(* IEC 61131-3 sources: AXOpen/src/components.rexroth.drives/ctrl/src/AxoCtrlxDriveXsc/TypesStructuresAndEnums, 22 files *)

(* ---- AxoCtrlxDriveXscErrorStruct.st ---- *)
NAMESPACE AXOpen.Components.Rexroth.Drives
    TYPE
        {S7.extern=ReadWrite}
        AxoCtrlxDriveXscErrorStruct :
        STRUCT
            Table       : AXOpen.Components.Rexroth.Drives.eAxoCtrlxDriveXscErrorTable;          (* Additional diagnosis table           *)
            Additional1 : DWORD;                (* Additional diagnosis number1         *)
            Additional2 : DWORD;                (* Additional diagnosis number2         *)
        END_STRUCT;
    END_TYPE
END_NAMESPACE

(* ---- eAxoCtrlxDriveXscErrorCode.st ---- *)
NAMESPACE AXOpen.Components.Rexroth.Drives
    TYPE PUBLIC
        eAxoCtrlxDriveXscErrorCode : WORD
        (
            NONE_ERROR                  := WORD#16#0000,     (* No error code available              *)
            (*                  invalid input                                                   *)
            INPUT_INVALID_ERROR         := WORD#16#0001,     (* Invalid input                        *)
            (*                  communications error                                            *)
            COMMUNICATION_ERROR         := WORD#16#0002,     (* Error while communication            *)
            (*                  data processing error                                           *)
            RESOURCE_ERROR              := WORD#16#0003,     (* Resource error                       *)
            ACCESS_ERROR                := WORD#16#0004,     (* Access error                         *)
            STATE_MACHINE_ERROR         := WORD#16#0005,     (* Invalid state State - Machine        *)
            INPUT_RANGE_ERROR           := WORD#16#0006,     (* Error because Input out of range     *)
            CALCULATION_ERROR           := WORD#16#0007,     (* Error while calculation              *)
            (*                  device error                                                    *)
            DEVICE_ERROR                := WORD#16#0008,     (* Device Error occurred                *)
            (*                  other error                                                     *)
            OTHER_ERROR                 := WORD#16#7FFE,     (* Undefined Error                      *)
            (*                  system error                                                    *)
            SYSTEM_ERROR                := WORD#16#7FFF      (* System error occured                 *)

                );
    END_TYPE
END_NAMESPACE

(* ---- eAxoCtrlxDriveXscErrorTable.st ---- *)
NAMESPACE AXOpen.Components.Rexroth.Drives
    TYPE PUBLIC
        eAxoCtrlxDriveXscErrorTable : WORD
        (
            NO_TABLE_USED           := WORD#16#0000,         //reserved
            SERCOS_TABLE            := WORD#16#0010,         //Sercos Error: Addtitional1 = Sercos Code
            MLDS_TABLE              := WORD#16#0020,         //Drive-based Motion - Logic
            MLC_TABLE               := WORD#16#0030,         //Controller - based Motion - Logic
            MTX_TABLE               := WORD#16#0040,         //CNC
            MLP_TABLE               := WORD#16#0050,         //PC  - based Motion Logic
            PLC_TABLE               := WORD#16#0060,         //PLC
            INDRV_TABLE             := WORD#16#0070,         //IndraDrive
            DIAX_TABLE              := WORD#16#0080,         //DIAX
            ECO_TABLE               := WORD#16#0090,         //EcoDrive
            PB_DP_TABLE             := WORD#16#0130,         //Profibus
            DEVICENET_TABLE         := WORD#16#0140,         //DeviceNet
            ETHERNET_TABLE          := WORD#16#0150,         //Ethernet
            INTERBUS_TABLE          := WORD#16#0160,         //Interbus
            F_RELATED_TABLE         := WORD#16#0170,         //function related
            USER1_TABLE             := WORD#16#1000,         //free User Table
            USER2_TABLE             := WORD#16#1001,         //free User Table
            USER3_TABLE             := WORD#16#1002,         //free User Table
            USER4_TABLE             := WORD#16#1003,         //free User Table
            USER5_TABLE             := WORD#16#1004,         //free User Table
            USER6_TABLE             := WORD#16#1005,         //free User Table
            USER7_TABLE             := WORD#16#1006,         //free User Table
            USER8_TABLE             := WORD#16#1007,         //free User Table
            USER9_TABLE             := WORD#16#1008,         //free User Table
            USER10_TABLE            := WORD#16#1009          //free User Table
        );
    END_TYPE
END_NAMESPACE

(* ---- AxoCtrlxDriveXsc_Component_Status.st ---- *)
NAMESPACE AXOpen.Components.Rexroth.Drives
    {S7.extern=ReadWrite}
    {#ix-attr:[Container(Layout.Stack)]}
    CLASS PUBLIC AxoCtrlxDriveXsc_Component_Status EXTENDS AXOpen.Components.Abstractions.AxoComponent_Status
        VAR PUBLIC

        END_VAR
    END_CLASS
END_NAMESPACE

(* ---- AxoCtrlxDriveXsc_Config.st ---- *)
NAMESPACE AXOpen.Components.Rexroth.Drives
    {S7.extern=ReadWrite}
    {#ix-attr:[Container(Layout.Stack)]}
    CLASS PUBLIC AxoCtrlxDriveXsc_Config
        VAR PUBLIC
            {#ix-set:AttributeName = "<#Info time#>"}
            InfoTime : LTIME := LT#5S;
            {#ix-set:AttributeName = "<#Error time#>"}
            ErrorTime : LTIME := LT#10S;
        END_VAR
    END_CLASS
END_NAMESPACE

(* ---- AxoCtrlxDriveXsc_Control.st ---- *)
NAMESPACE AXOpen.Components.Rexroth.Drives
    {S7.extern=ReadWrite}
    {#ix-attr:[Container(Layout.Stack)]}
    CLASS PUBLIC AxoCtrlxDriveXsc_Control
        VAR PUBLIC

        END_VAR
    END_CLASS
END_NAMESPACE

(* ---- AxoCtrlxDriveXsc_In.st ---- *)
NAMESPACE AXOpen.Components.Rexroth.Drives
    {S7.extern=ReadWrite}
    {#ix-attr:[Container(Layout.Wrap)]}
    CLASS PUBLIC AxoCtrlxDriveXsc_In
        VAR PUBLIC
            {#ix-set:AttributeName = "<#Status#>"}
            {#ix-attr:[ReadOnly()]}
            Status           :   AxoCtrlxDriveXsc_Status;
        END_VAR
    END_CLASS
END_NAMESPACE

(* ---- AxoCtrlxDriveXsc_Out.st ---- *)
NAMESPACE AXOpen.Components.Rexroth.Drives
    {S7.extern=ReadWrite}
    {#ix-attr:[Container(Layout.Wrap)]}
    CLASS PUBLIC AxoCtrlxDriveXsc_Out
        VAR PUBLIC
            {#ix-set:AttributeName = "<#Control#>"}
            {#ix-attr:[ReadOnly()]}
            Control           :   AxoCtrlxDriveXsc_Control;
        END_VAR
    END_CLASS
END_NAMESPACE

(* ---- AxoCtrlxDriveXsc_Status.st ---- *)
NAMESPACE AXOpen.Components.Rexroth.Drives
    {S7.extern=ReadWrite}
    {#ix-attr:[Container(Layout.Stack)]}
    CLASS PUBLIC AxoCtrlxDriveXsc_Status
        VAR PUBLIC

        END_VAR
    END_CLASS
END_NAMESPACE

(* ---- AxoCtrlxDriveXscAxisData.st ---- *)
NAMESPACE AXOpen.Components.Rexroth.Drives
    {S7.extern=ReadWrite}
    CLASS AxoCtrlxDriveXscAxisData
        VAR PUBLIC
            (* Commands *)
            CallAxis					:	BOOL;			//Call axis method for cyclic communication
            ReadOnlyData				:	BOOL;			//Read only data values from drive
            CallNumberCyclic			:	INT :=-1; 		//Number of method call's for cyclic communication
            WriteCommand				:	BOOL;			//Write command to drive
            PowerOnReq					:	BOOL;			//Request to power the drive on
            ResetReq					:	BOOL;			//Request to reset the drive
            HomingReq					:	BOOL;			//Request to start homing
            JogPositiveReq				:	BOOL;			//Request to jog the drive in positive direction
            JogNegativeReq				:	BOOL;			//Request to jog the drive in negative direction
            DriveStopReq				:	BOOL;			//Set Drive Stop with writing deceleration value to drive
            DriveHaltReq				:	BOOL;			//Set Drive Halt with writing deceleration value to drive
            MoveVelocityReq				:	BOOL;			//Command is velocity
            TorqueControlReq				:	BOOL;			//Command is torque
            Relative					:	BOOL; 			//Move relative to (last recommended) positioning command value
            Additive					:	BOOL; 			//Move additive to actual position; works only if relative possitioning active
            Position					:	LREAL;			//Target position for the motion  (negative or positive)
            Velocity					:	LREAL;			//Value of the maximum velocity (always positive) (not necessarily reached) [u/s].
            Acceleration				:	LREAL;			//Value of the acceleration (always positive) (increasing energy of the motor) [u/s2]
            Deceleration				:	LREAL;			//Value of the deceleration (always positive) (decreasing energy of the motor) [u/s2]
            Jerk						:	LREAL;			//Value of the jerk (always positive) [u/s3]
            Torque						:	LREAL;			//Value of the torque (always positive)
            S_0_0144_SignalStateWord	: 	WORD;			//S-0-0144 SignalStateWord*)
            CallAxisParameterMethod		:	BOOL;			//Call axis method for parameter read/write
            EnableAcyclicCommunication	:	BOOL;			//Enable acyclic communication (for parameter read/write)
            CallNumberAcyclic			:	INT;			//Number of method call's for acyclic communication
            WriteParameter				:	BOOL;			//FALSE = read, TRUE  = write Value of selected Parameter
            SelectDataType				:	UINT;			//0= Bool, 1 = Any, 2 = REAL
            ParameterNumber				:	DINT;			//Parameter number
            WriteValueLint				:	LINT;			//DINT value to be written
            WriteValueReal				:	REAL;			//REAL value to be written
            OverrideVelocityFactor		:	LREAL := 1.0;	//LREAL value to be written
            OverrideAccelerationFactor	:	LREAL := 1.0;	//LREAL value to be written
            OverrideJerkFactor			:	LREAL := 1.0;	//LREAL value to be written
        (* States *)
            CommandWriteActive			:	BOOL; 			//Command transfer to drive is active
            SetpointReached				: 	BOOL;			//Setpoint reached
            PowerOK						:	BOOL; 			//Power OK
            HomeOK						:	BOOL;			//Drive has reached the homeposition
            ResetOK						:	BOOL; 			//Reset done
            HomingRunning				:	BOOL;			//Homing is active
            Stopped						:	BOOL; 			//Drive in stopped regularly
            Standstill					:	BOOL; 			//Drive in standstill
            InPosition					:	BOOL; 			//Drive in position
            StoppedDueError				:	BOOL; 			//Drive in stop due to error
            MessageActive				:	BOOL;			//Class 3 diagnostics (message) present
            WarningActive				:	BOOL;			//Class 2 diagnostics (warning) present
            FailureActive				:	BOOL;			//Class 1 diagnostics (failure) present
            PowerError					:	BOOL; 			//Power-Failure
            StopError					:	BOOL;			//Stopping-Failure
            ContinuousMotion			:	BOOL; 			//Continius motion
            DiscreteMotion				:	BOOL; 			//Discrete motion
            SynchronizedMotion			:	BOOL;			//Synchronized motion
            Error						:	BOOL;			//Error
            ErrorID						:	AXOpen.Components.Rexroth.Drives.eAxoCtrlxDriveXscErrorCode;		//Error identification, ErrorCode
            ErrorIdent					:	AXOpen.Components.Rexroth.Drives.AxoCtrlxDriveXscErrorStruct;	//Error identification
            ActualPosition				:	LREAL; 			//Shows actual position
            ActualVelocity				:	LREAL; 			//Shows actual velocity
            ActualTorque				:	LREAL; 			//Shows actual torque
            CheckAccessOK				:	BOOL := TRUE;	//Flag for checking valid access at Axis_Data array
            S_0_0145_SignalControlWord	:	WORD;			//S-0-0145 wSignalControlWord, **** exept bit 0 *****)

            DoneAcyclicCommunication 	:	BOOL; 			//Reading/writing of the individual parameter completed, output variables valid
            ActiveAcyclicCommunication	: 	BOOL; 			//Reading/writing of the individual parameter active, output variables invalid
            DecimalPlaces 				:	UINT;			//Decimal places of the selected parameters
            DataTypeRead				:	UINT; 			//Read data type of the selected parameters
            DataLengthRead				:	UINT;			//Length of the read parameters
            ReadValueDint				:	DINT;			//DINT Operating value of the individual parameter without weighting
            ReadValueReal				:	REAL;			//REAL weighted operating value
            Error_AcyclicCommunication	:	BOOL := FALSE;  //Error
            ErrorID_AcyclicCommunication:   AXOpen.Components.Rexroth.Drives.eAxoCtrlxDriveXscErrorCode;		//Error identification, ErrorCode
            ErrorIdent_AcyclicCommunication:AXOpen.Components.Rexroth.Drives.AxoCtrlxDriveXscErrorStruct; 	//Error identification
            hwID                :   WORD;
            hwIdParamCh_IDN     :   WORD;
            hwIdInput_9_Words   :   WORD;
            hwIdOutput_13_Words :   WORD;
        END_VAR
    END_CLASS
END_NAMESPACE

(* ---- AxoCtrlxDriveXscAxisReference.st ---- *)
// USING AXOpen.Components.Drives;

NAMESPACE AXOpen.Components.Rexroth.Drives
    {S7.extern=ReadWrite}
    CLASS AxoCtrlxDriveXscAxisReference IMPLEMENTS AXOpen.Components.Abstractions.Drives.IAxoAxisReference
        VAR PUBLIC
            FieldBus_In     :   AXOpen.Components.Rexroth.Drives.AxoCtrlxDriveXscFieldBusIn;
            FieldBus_Out    :   AXOpen.Components.Rexroth.Drives.AxoCtrlxDriveXscFieldBusOut;
            Parameter_In    :   AXOpen.Components.Rexroth.Drives.AxoCtrlxDriveXscParameterIn;
            Parameter_Out   :   AXOpen.Components.Rexroth.Drives.AxoCtrlxDriveXscParameterOut;
            Data            :   AXOpen.Components.Rexroth.Drives.AxoCtrlxDriveXscAxisData;
            Config          :   AXOpen.Components.Drives.AxoDrive_Config;
            Status          :   AXOpen.Components.Drives.AxoDrive_Status;
        END_VAR
    END_CLASS
END_NAMESPACE

(* ---- AxoCtrlxDriveXscDriveControlWord_S_0_0134_0_0.st ---- *)
NAMESPACE AXOpen.Components.Rexroth.Drives
    {S7.extern=ReadWrite}
    {#ix-attr:[Container(Layout.Wrap)]}
    {#ix-attr:[Group(GroupLayout.GroupBox)]}
    {#ix-set:AttributeName = "<#DriveControlWord#>"}
    CLASS AxoCtrlxDriveXscDriveControlWord_S_0_0134_0_0
        VAR PUBLIC
            {#ix-set:AttributeName = "<#_bit00_Reserve#>"}
            {#ix-attr:[ReadOnly()]}
            _bit00_Reserve 				:	BOOL;
            {#ix-set:AttributeName = "<#_bit01_Reserve#>"}
            {#ix-attr:[ReadOnly()]}
            _bit01_Reserve 				:	BOOL;
            {#ix-set:AttributeName = "<#_bit02_Reserve#>"}
            {#ix-attr:[ReadOnly()]}
            _bit02_Reserve 				:	BOOL;
            {#ix-set:AttributeName = "<#_bit03_Reserve#>"}
            {#ix-attr:[ReadOnly()]}
            _bit03_Reserve 				:	BOOL;
            {#ix-set:AttributeName = "<#_bit04_Reserve#>"}
            {#ix-attr:[ReadOnly()]}
            _bit04_Reserve 				:	BOOL;
            {#ix-set:AttributeName = "<#_bit05_Reserve#>"}
            {#ix-attr:[ReadOnly()]}
            _bit05_Reserve 				:	BOOL;
            {#ix-set:AttributeName = "<#_bit06_Reserve#>"}
            {#ix-attr:[ReadOnly()]}
            _bit06_Reserve 				:	BOOL;
            {#ix-set:AttributeName = "<#_bit07_Reserve#>"}
            {#ix-attr:[ReadOnly()]}
            _bit07_Reserve 				:	BOOL;

            {#ix-set:AttributeName = "<#Command operation mode Bit 0#>"}
            {#ix-attr:[ReadOnly()]}
            CommandOperationModeBit0 	:	BOOL;		//  Command operation mode bit 0                        |   000:  Primary operation mode
                                                        //                                                      |   001:  Secondary operation mode 1
            {#ix-set:AttributeName = "<#Command operation mode Bit 1#>"}
            {#ix-attr:[ReadOnly()]}
            CommandOperationModeBit1 	:	BOOL;		//  Command operation mode bit 1                        |   010:  Secondary operation mode 2
                                                        //                                                      |   011:  Secondary operation mode 3
                                                        //                                                      |   100:  Secondary operation mode 4
            {#ix-set:AttributeName = "<#Command operation mode Bit 2#>"}
            {#ix-attr:[ReadOnly()]}
            CommandOperationModeBit2 	:	BOOL;		//  Command operation mode bit 2                        |   101:  Secondary operation mode 5
                                                        //                                                      |   110:  Secondary operation mode 6
                                                        //                                                      |   111:  Secondary operation mode 7
            {#ix-set:AttributeName = "<#_bit11_Reserve#>"}
            {#ix-attr:[ReadOnly()]}
            _bit11_Reserve 				:	BOOL;
            {#ix-set:AttributeName = "<#_bit12_Reserve#>"}
            {#ix-attr:[ReadOnly()]}
            _bit12_Reserve 				:	BOOL;
            {#ix-set:AttributeName = "<#Drive Halt#>"}
            {#ix-attr:[ReadOnly()]}
            DriveHalt 				:	BOOL;		        //  1-0 change: Deceleration of drive while maintaining maximum acceleration (S‑0‑0138 - only possible if bits 14 and 15 = 1)
            {#ix-set:AttributeName = "<#Drive enable#>"}
            {#ix-attr:[ReadOnly()]}
            DriveEnable 				:	BOOL;		    //  Negative edge: Torque disable without delay (independent of bit 15 or 13)
            {#ix-set:AttributeName = "<#Drive On#>"}
            {#ix-attr:[ReadOnly()]}
            DriveOn 				:	BOOL;		        //  Negative edge: Best possible deceleration (only possible if bit 14 = 1)
        END_VAR
    END_CLASS
END_NAMESPACE

(* ---- AxoCtrlxDriveXscDriveStatusWord_S_0_0135_0_0.st ---- *)
NAMESPACE AXOpen.Components.Rexroth.Drives
    {S7.extern=ReadWrite}
    {#ix-attr:[Container(Layout.Wrap)]}
    {#ix-attr:[Group(GroupLayout.GroupBox)]}
    {#ix-set:AttributeName = "<#DriveStatusWord#>"}
    CLASS AxoCtrlxDriveXscDriveStatusWord_S_0_0135_0_0
        VAR PUBLIC
            {#ix-set:AttributeName = "<#_bit00_Reserve#>"}
            // {#ix-attr:[ReadOnly()]}
            _bit00_Reserve 				:	BOOL;
            {#ix-set:AttributeName = "<#_bit01_Reserve#>"}
            // {#ix-attr:[ReadOnly()]}
            _bit01_Reserve 				:	BOOL;
            {#ix-set:AttributeName = "<#_bit02_Reserve#>"}
            // {#ix-attr:[ReadOnly()]}
            _bit02_Reserve 				:	BOOL;
            {#ix-set:AttributeName = "<#CommandProcessingStatus#>"}
            // {#ix-attr:[ReadOnly()]}
            CommandProcessingStatus		:	BOOL;		//  0 - Drive ignores command value input           |   1 -Drive follows command value input
            {#ix-set:AttributeName = "<#InStandstill#>"}
            // {#ix-attr:[ReadOnly()]}
            InStandstill 				:	BOOL;		//  Drive "Halt" status                             |   1- Act vel < standstill window
            {#ix-set:AttributeName = "<#InReference#>"}
            // {#ix-attr:[ReadOnly()]}
            InReference 				:	BOOL;		//  Drive hommed
            {#ix-set:AttributeName = "<#_bit06_Reserve#>"}
            // {#ix-attr:[ReadOnly()]}
            _bit06_Reserve 				:	BOOL;
            {#ix-set:AttributeName = "<#HardwareLock#>"}
            // {#ix-attr:[ReadOnly()]}
            HardwareLock                :	BOOL;       //  Hardware lock (E-stop)
            {#ix-set:AttributeName = "<#ActualOperatingModeBit0#>"}
            // {#ix-attr:[ReadOnly()]}
            ActualOperatingModeBit0 	:	BOOL;		//  Actual_operating mode bit 0                     |   000:  Primary operation mode
                                                        //                                                  |   001:  Secondary operation mode 1
            {#ix-set:AttributeName = "<#ActualOperatingModeBit1#>"}
            // {#ix-attr:[ReadOnly()]}
            ActualOperatingModeBit1 	:	BOOL;		//  Actual_operating mode bit 1                     |   010:  Secondary operation mode 2
                                                        //                                                  |   011:  Secondary operation mode 3
                                                        //                                                  |   100:  Secondary operation mode 4
            {#ix-set:AttributeName = "<#ActualOperatingModeBit2#>"}
            // {#ix-attr:[ReadOnly()]}
            ActualOperatingModeBit2 	:	BOOL;		//  Actual_operating mode bit 2                     |   101:  Secondary operation mode 5
                                                        //                                                  |   110:  Secondary operation mode 6
                                                        //                                                  |   111:  Secondary operation mode 7
            {#ix-set:AttributeName = "<#_bit11_Reserve#>"}
            // {#ix-attr:[ReadOnly()]}
            _bit11_Reserve 				:	BOOL;
            {#ix-set:AttributeName = "<#WarningZKL2#>"}
            // {#ix-attr:[ReadOnly()]}
            WarningZKL2 				:	BOOL;		//  Warning ZKL2
            {#ix-set:AttributeName = "<#DriveErrorZKL1#>"}
            // {#ix-attr:[ReadOnly()]}
            DriveErrorZKL1 				:	BOOL;		//  Drive Error ZKL1
            {#ix-set:AttributeName = "<#ReadyForOperation Bit 0#>"}
            // {#ix-attr:[ReadOnly()]}
            ReadyForOperationBit0       :	BOOL;		//  Ready to operate bit 0 lower significant bit    |   10: Control section and power section ready for op. (Ab)
                                                        //                                                  |   11: In operation, with torque (e.g. AF)
            {#ix-set:AttributeName = "<#ReadyForOperation Bit 1#>"}
            // {#ix-attr:[ReadOnly()]}
            ReadyForOperationBit1       :	BOOL;		//  Ready to operate bit 1 higher significant bit   |   00: Not ready for power on (e.g., P2)
                                                        //                                                  |   01: Ready for power on (bb)
        END_VAR
    END_CLASS
END_NAMESPACE

(* ---- AxoCtrlxDriveXscFieldBusIn.st ---- *)
NAMESPACE AXOpen.Components.Rexroth.Drives
    {S7.extern=ReadWrite}
    CLASS AxoCtrlxDriveXscFieldBusIn
        (******************* Drive configuration  ***********************
        Master communication; Fieldbus settings:
                Parameter channel 10Bytes / 5 Words I/O
                Parameter channel: F-Modul not used
                Realtime Input channel 18Bytes / 9 Words I/O
                Realtime Output channel 26Bytes / 13 Words I/O
                Profile type: * free configurable mode*
                    Configuration of realtime channel:
                        realtime input (configured feedback values):	    (9words)
                                P-0-4078 Fieldbus status WORD               (2bytes)
                                S-0-0051 Position feedback 1 value          (4bytes)
                                S-0-0040 Veloccity feedback value           (4bytes)
                                S-0-0390 Diagnostig message number          (4bytes)
                                S-0-0144 Signal status  word			    (2bytes)
                                S-0-0084 Actual torque/force value          (2bytes)
                        realtime output (configured command values):		(13words)
                                P-0-4077 Fieldbus control WORD              (2bytes)
                                S-0-0282 Positioning command value          (4bytes)
                                S-0-0259 Positioning velocity value         (4bytes)
                                S-0-0260 Positioning Accelelration          (4bytes)
                                S-0-0359 Positioning Deceleration           (4bytes)
                                S-0-0145 Signal control word                (2bytes)
                                S-0-0080 Torque/force command value		    (2bytes)
                                S-0-0193 Positioning jerk                   (4bytes)
                General settings:
                        S-0-0027, Configuration list signal control word -> Number 0; Content S-0-0393
                        S-0-0329, Assign list signal control word -> Number 0; Content 2
                        Primary operation mode: Drive controlled positioning, encoder 1 (without axis control word)
                        Secondary operation mode: Torque/force control
        *)
        VAR PUBLIC
            PhaseAcknowledgeBit0		:	BOOL;		//Operating mode acknowledge bit 0
            PhaseAcknowledgeBit1 		:	BOOL;		//Operating mode acknowledge bit 1
            InReference 				:	BOOL;		//In reference
            InStandstill 				:	BOOL;		//In standstill
            SetpointReached				:	BOOL;		//Setpoint reached
            CommandChangeBit 			:	BOOL;		//Command change bit
            OperatingModeError 			:	BOOL;		//Operating mode_error
            StatusSetpointProcess 		:	BOOL;		//Status setpoint processing
            ActualOperatingModeBit0 	:	BOOL;		//Actual_operating mode bit 0
            ActualOperatingModeBit1 	:	BOOL;		//Actual_operating mode bit 1
            SetpointAcknowledge 		:	BOOL;		//Setpoint acknowledge
            MessageZKL3 				:	BOOL;		//Message ZKL3
            WarningZKL2 				:	BOOL;		//Warning ZKL2
            DriveErrorZKL1 				:	BOOL;		//Drive Error ZKL1
            ReadyToOperateBit0 			:	BOOL;		//Ready to operate bit 0
            ReadyToOperateBit1 			:	BOOL;		//Ready to operate bit 1
            S_0_0051_ActualPosition		:	DWORD;		//Actual position
            S_0_0040_ActualVelocity		:	DWORD;		//Actual velocity
            S_0_0390_Diagnosis			:	DWORD;		//Diagnosis
            S_0_0144_SignalStatusWord	:	WORD;		//Signal status word
            S_0_0084_ActualTorque 		:	WORD;		//Actual torque
        END_VAR
    END_CLASS

END_NAMESPACE

(* ---- AxoCtrlxDriveXscFieldBusOut.st ---- *)
NAMESPACE AXOpen.Components.Rexroth.Drives
    {S7.extern=ReadWrite}
    CLASS AxoCtrlxDriveXscFieldBusOut
        (******************* Drive configuration  ***********************
        Master communication; Fieldbus settings:
                Parameter channel 10Bytes / 5 Words I/O
                Parameter channel: F-Modul not used
                Realtime Input channel 18Bytes / 9 Words I/O
                Realtime Output channel 26Bytes / 13 Words I/O
                Profile type: * free configurable mode*
                    Configuration of realtime channel:
                        realtime input (configured feedback values):	    (9words)
                                P-0-4078 Fieldbus status WORD               (2bytes)
                                S-0-0051 Position feedback 1 value          (4bytes)
                                S-0-0040 Veloccity feedback value           (4bytes)
                                S-0-0390 Diagnostig message number          (4bytes)
                                S-0-0144 Signal status  word			    (2bytes)
                                S-0-0084 Actual torque/force value          (2bytes)
                        realtime output (configured command values):		(13words)
                                P-0-4077 Fieldbus control WORD              (2bytes)
                                S-0-0282 Positioning command value          (4bytes)
                                S-0-0259 Positioning velocity value         (4bytes)
                                S-0-0260 Positioning Accelelration          (4bytes)
                                S-0-0359 Positioning Deceleration           (4bytes)
                                S-0-0145 Signal control word                (2bytes)
                                S-0-0080 Torque/force command value		    (2bytes)
                                S-0-0193 Positioning jerk                   (4bytes)
                General settings:
                        S-0-0027, Configuration list signal control word -> Number 0; Content S-0-0393
                        S-0-0329, Assign list signal control word -> Number 0; Content 2
                        Primary operation mode: Drive controlled positioning, encoder 1 (without axis control word)
                        Secondary operation mode: Torque/force control
        *)
        VAR PUBLIC
            SetpointAcceptance 				:	BOOL;			//Setpoint acceptance
            OperatingModeSet 				:	BOOL;			//Operating mode set
            DriveToZeroPoint 				:	BOOL;			//Drive to zero point
            AbsoluteRelative 				:	BOOL;			//Position absolute = 0 or relative = 1
            ImmediateBlockChange 			:	BOOL;			//Immediate change
            ErrorDelete 					:	BOOL;			//Clear error
            JogForward 						:	BOOL;			//Jog forward
            JogBackward 					:	BOOL;			//Jog backward
            SetOperatingModeBit0 			:	BOOL;			//Setpoint operating mode_bit0
            SetOperatingModeBit1 			:	BOOL;			//Setpoint operating mode_bit1
            Iposync 						:	BOOL;			//Only in cycl. pos. control
            DriveHalt 						:	BOOL;			//Drive halt
            DriveEnable 					:	BOOL;			//Drive enable
            DriveOn 						:	BOOL;			//Drive on
            S_0_0282_CommandPosition		: 	DWORD;			//Command position
            S_0_0259_CommandVelocity		: 	DWORD;          //Command velocity
            S_0_0260_CommandAcceleration	: 	DWORD;          //Command acceleration
            S_0_0359_CommandDecceleration	: 	DWORD;          //Command decceleration
            S_0_0145_SignalControlWord		: 	WORD;           //Signal control word
            S_0_0080_TorqueForceCommand     :   WORD;           //Torque/force command value
            S_0_0193_CommandJerk            :   DWORD;          //Command jerk
        END_VAR
    END_CLASS
END_NAMESPACE

(* ---- AxoCtrlxDriveXscHWIDs.st ---- *)
NAMESPACE AXOpen.Components.Rexroth.Drives
   {S7.extern=ReadWrite}
	CLASS AxoCtrlxDriveXscHWIDs
      VAR PUBLIC
         {#ix-set:AttributeName = "<#Hardware ID Device#>"}
         HW_Device            : UINT;
         {#ix-set:AttributeName = "<#Hardware ID 'Outputs' module#>"}
         HW_Outputs           : UINT;
         {#ix-set:AttributeName = "<#Hardware ID 'Inputs' module#>"}
         HW_Inputs            : UINT;
         {#ix-set:AttributeName = "<#Hardware ID 'S_0_0134_0_0__Servodrive_profile__Control_word' submodule#>"}
         HW_S_0_0134_0_0      : UINT;
         {#ix-set:AttributeName = "<#Hardware ID 'S_0_0145_0_0__Signal_control_word__Value' submodule#>"}
         HW_S_0_0145_0_0      : UINT;
         {#ix-set:AttributeName = "<#Hardware ID 'S_0_0282_0_0__Drive_controlled_positioning__Command_value' submodule#>"}
         HW_S_0_0282_0_0      : UINT;
         {#ix-set:AttributeName = "<#Hardware ID 'S_0_0259_0_0__Positioning_profile__Profile_velocity' submodule#>"}
         HW_S_0_0259_0_0      : UINT;
         {#ix-set:AttributeName = "<#Hardware ID 'S_0_0260_0_0__Positioning_profile__Acceleration' submodule#>"}
         HW_S_0_0260_0_0      : UINT;
         {#ix-set:AttributeName = "<#Hardware ID 'S_0_0359_0_0__Positioning_profile__Deceleration' submodule#>"}
         HW_S_0_0359_0_0      : UINT;
         {#ix-set:AttributeName = "<#Hardware ID 'S_0_1720_0_1__Power_supply_control__Control_word' submodule#>"}
         HW_S_0_1720_0_1      : UINT;
         {#ix-set:AttributeName = "<#Hardware ID 'S_0_0092_0_0__Torque_force_limitation__Limit_value_bipolar' submodule#>"}
         HW_S_0_0092_0_0      : UINT;
         {#ix-set:AttributeName = "<#Hardware ID 'S_0_0080_0_0__Torque_force_command_value' submodule#>"}
         HW_S_0_0080_0_0      : UINT;
         {#ix-set:AttributeName = "<#Hardware ID 'S_0_0193_0_0__Positioning_jerk' submodule#>"}
         HW_S_0_0193_0_0      : UINT;
         {#ix-set:AttributeName = "<#Hardware ID 'S_0_0135_0_0__Servodrive_profile__Status_word' submodule#>"}
         HW_S_0_0135_0_0      : UINT;
         {#ix-set:AttributeName = "<#Hardware ID 'S_0_0144_0_0__Signal_status_word__Value' submodule#>"}
         HW_S_0_0144_0_0      : UINT;
         {#ix-set:AttributeName = "<#Hardware ID 'S_0_0386_0_0__Position_controller__Position_actual_value' submodule#>"}
         HW_S_0_0386_0_0      : UINT;
         {#ix-set:AttributeName = "<#Hardware ID 'S_0_0535_0_0__Velocity_controller__Velocity_actual_value' submodule#>"}
         HW_S_0_0535_0_0      : UINT;
         {#ix-set:AttributeName = "<#Hardware ID 'S_0_0390_0_0__Diagnostic_message__Manufacturer_status_register' submodule#>"}
         HW_S_0_0390_0_0      : UINT;
         {#ix-set:AttributeName = "<#Hardware ID 'S_0_1720_0_2__Power_supply_control__Status_word' submodule#>"}
         HW_S_0_1720_0_2      : UINT;
         {#ix-set:AttributeName = "<#Hardware ID 'S_0_0084_0_0__Torque_force_feedback_value' submodule#>"}
         HW_S_0_0084_0_0      : UINT;
         {#ix-set:AttributeName = "<#Hardware ID 'P_0_0106_0_0__STO_function__Operating_status' submodule#>"}
         HW_P_0_0106_0_0      : UINT;
      END_VAR
   END_CLASS
END_NAMESPACE

(* ---- AxoCtrlxDriveXscParameterIn.st ---- *)
NAMESPACE AXOpen.Components.Rexroth.Drives
    {S7.extern=ReadWrite}
    CLASS AxoCtrlxDriveXscParameterIn
        (******************* Drive configuration  ***********************
        Master communication; Fieldbus settings:
                Parameter channel 10Bytes / 5 Words I/O
                Parameter channel: F-Modul not used
                Realtime Input channel 18Bytes / 9 Words I/O
                Realtime Output channel 26Bytes / 13 Words I/O
                Profile type: * free configurable mode*
                    Configuration of realtime channel:
                        realtime input (configured feedback values):	    (9words)
                                P-0-4078 Fieldbus status WORD               (2bytes)
                                S-0-0051 Position feedback 1 value          (4bytes)
                                S-0-0040 Veloccity feedback value           (4bytes)
                                S-0-0390 Diagnostig message number          (4bytes)
                                S-0-0144 Signal status  word			    (2bytes)
                                S-0-0084 Actual torque/force value          (2bytes)
                        realtime output (configured command values):		(13words)
                                P-0-4077 Fieldbus control WORD              (2bytes)
                                S-0-0282 Positioning command value          (4bytes)
                                S-0-0259 Positioning velocity value         (4bytes)
                                S-0-0260 Positioning Accelelration          (4bytes)
                                S-0-0359 Positioning Deceleration           (4bytes)
                                S-0-0145 Signal control word                (2bytes)
                                S-0-0080 Torque/force command value		    (2bytes)
                                S-0-0193 Positioning jerk                   (4bytes)
                General settings:
                        S-0-0027, Configuration list signal control word -> Number 0; Content S-0-0393
                        S-0-0329, Assign list signal control word -> Number 0; Content 2
                        Primary operation mode: Drive controlled positioning, encoder 1 (without axis control word)
                        Secondary operation mode: Torque/force control
        *)
        VAR PUBLIC
            Datalength	:	BYTE;	//Length of  transfer data*)
            FL_0		:	BOOL;	//Length userdata bit 0
            FL_1		:	BOOL;	//Length userdata bit 1
            FL_2		:	BOOL;	//Length userdata bit 2
            FL_3		:	BOOL;	//Length userdata bit 3
            ToggleBit	:	BOOL;	//Toggle bit
            LastBit		:	BOOL;	//Last bit
            Failure		:	BOOL;	//Failure while communication
            Reserve		:	BOOL;	//Reserve
            DataWord_0	:	WORD;	//Data WORD 0
            DataWord_1	:	WORD;	//Data word 1
            DataWord_2	:	WORD;	//Data word 2
            DataWord_3	:	WORD;	//Data word 3
        END_VAR
    END_CLASS
 END_NAMESPACE

(* ---- AxoCtrlxDriveXscParameterOut.st ---- *)
NAMESPACE AXOpen.Components.Rexroth.Drives
    {S7.extern=ReadWrite}
    CLASS AxoCtrlxDriveXscParameterOut
        (******************* Drive configuration  ***********************
        Master communication; Fieldbus settings:
                Parameter channel 10Bytes / 5 Words I/O
                Parameter channel: F-Modul not used
                Realtime Input channel 18Bytes / 9 Words I/O
                Realtime Output channel 26Bytes / 13 Words I/O
                Profile type: * free configurable mode*
                    Configuration of realtime channel:
                        realtime input (configured feedback values):	    (9words)
                                P-0-4078 Fieldbus status WORD               (2bytes)
                                S-0-0051 Position feedback 1 value          (4bytes)
                                S-0-0040 Veloccity feedback value           (4bytes)
                                S-0-0390 Diagnostig message number          (4bytes)
                                S-0-0144 Signal status  word			    (2bytes)
                                S-0-0084 Actual torque/force value          (2bytes)
                        realtime output (configured command values):		(13words)
                                P-0-4077 Fieldbus control WORD              (2bytes)
                                S-0-0282 Positioning command value          (4bytes)
                                S-0-0259 Positioning velocity value         (4bytes)
                                S-0-0260 Positioning Accelelration          (4bytes)
                                S-0-0359 Positioning Deceleration           (4bytes)
                                S-0-0145 Signal control word                (2bytes)
                                S-0-0080 Torque/force command value		    (2bytes)
                                S-0-0193 Positioning jerk                   (4bytes)
                General settings:
                        S-0-0027, Configuration list signal control word -> Number 0; Content S-0-0393
                        S-0-0329, Assign list signal control word -> Number 0; Content 2
                        Primary operation mode: Drive controlled positioning, encoder 1 (without axis control word)
                        Secondary operation mode: Torque/force control
        *)
        VAR PUBLIC
            Datalength		:	BYTE := BYTE#04;//Length of transfer data
            FL_0			:	BOOL;			//Length userdata bit 0
            FL_1			:	BOOL;			//Length userdata bit 1
            FL_2			:	BOOL;			//Length userdata bit 2
            FL_3			:	BOOL;			//Length userdata bit 3
            ToggleBit		:	BOOL;			//Toggle bit
            LastBit			:	BOOL;			//Last bit
            Initalisation	:	BOOL := TRUE;	//Initialisation
            Reserve			:	BOOL;			//Reserve
            Index			:	WORD;			//Index number
            Subindex		:	BYTE;			//Subindex number
            Axis			:	BYTE;			//Axis number
            DataWord_0		:	WORD;			//Data word 0
            DataWord_1		:	WORD;			//Data word 1
        END_VAR
    END_CLASS
END_NAMESPACE

(* ---- AxoCtrlxDriveXscSignalControlWord_S_0_0145_0_0.st ---- *)
NAMESPACE AXOpen.Components.Rexroth.Drives
    {S7.extern=ReadWrite}
    {#ix-attr:[Container(Layout.Wrap)]}
    {#ix-attr:[Group(GroupLayout.GroupBox)]}
    {#ix-set:AttributeName = "<#SignalControlWord#>"}
    CLASS AxoCtrlxDriveXscSignalControlWord_S_0_0145_0_0
        VAR PUBLIC
            {#ix-set:AttributeName = "<#Acceptance of positioning command value#>"}
            AcceptanceOfPositioningCommandValue:	BOOL;		                                    //  Bit 0 of the Drive-controlled positioning: Control word (S-0-0346) !!! must be set in drive !!!
            {#ix-set:AttributeName = "<#_bit01_Reserve#>"}
            _bit01_Reserve 				:	BOOL;
            {#ix-set:AttributeName = "<#Homing control#>"}
            HomingControl 				:	BOOL;		                                            //  Bit 0 of the Homing control: C0600 Command drive-controlled procedure (S-0-0148) !!! must be set in drive !!!
            {#ix-set:AttributeName = "<#Absolute/Relative type of positioning command value#>"}
            AbsoluteRelative 				:	BOOL;				                                //  Bit 3 of the Drive-controlled positioning: Control word (S-0-0346) !!! must be set in drive !!!
            {#ix-set:AttributeName = "<#Immediate block change#>"}
            ImmediateChange 				:	BOOL;                                               //  Bit 5 of the Drive-controlled positioning: Control word (S-0-0346) !!! must be set in drive !!!
            {#ix-set:AttributeName = "<#Clear error#>"}
            ClearError  :	BOOL;                                                                   //  Bit 0 of the Class 1 diagnostics: C0500 Reset command (S-0-0099) !!! must be set in drive !!!
            {#ix-set:AttributeName = "<#Infinite travel in positive direction (jog+)#>"}
            JogPositive :	BOOL;                                                                   //  Bit 1 of the Drive-controlled positioning: Control word (S-0-0346) !!! must be set in drive !!!
            {#ix-set:AttributeName = "<#Infinite travel in negative direction (jog-)#>"}
            JogNegative :	BOOL;                                                                   //  Bit 2 of the Drive-controlled positioning: Control word (S-0-0346) !!! must be set in drive !!!
            {#ix-set:AttributeName = "<#Activate configuration mode#>"}
            SwitchToCM  :	BOOL;                                                                   //  Bit 0 of the Subdevice STM: C0400 Activate configuration mode (S-0-0420) !!! must be set in drive !!!
            {#ix-set:AttributeName = "<#Activate operation mode#>"}
            SwitchTo0M  :	BOOL;                                                                   //  Bit 0 of the Subdevice STM: C0200 Activate operation mode (S-0-0422) !!! must be set in drive !!!
            {#ix-set:AttributeName = "<#CancelReferencePoint#>"}
            CancelReferencePoint        :	BOOL;		                                            // Homing function: C1500 Command cancel reference point (0x2500:01 / S-0-0191 / --) !!! must be set in drive !!!
            {#ix-set:AttributeName = "<#Device reboot#>"}
            DeviceReboot 				:	BOOL;
            {#ix-set:AttributeName = "<#_bit12_Reserve#>"}
            _bit12_Reserve 				:	BOOL;
            {#ix-set:AttributeName = "<#_bit13_Reserve#>"}
            _bit13_Reserve 				:	BOOL;
            {#ix-set:AttributeName = "<#_bit14_Reserve#>"}
            _bit14_Reserve 				:	BOOL;
            {#ix-set:AttributeName = "<#Set absolute position function#>"}
            SetAbsPositionFunction  :	BOOL;                                                       //  Bit 0 of the Set absolute position function: C0300 Command procedure (S-0-0447) !!! must be set in drive !!!
        END_VAR
    END_CLASS
END_NAMESPACE

(* ---- AxoCtrlxDriveXscSignalStatusWord_S_0_0144_0_0.st ---- *)
NAMESPACE AXOpen.Components.Rexroth.Drives
    {S7.extern=ReadWrite}
    {#ix-attr:[Container(Layout.Wrap)]}
    {#ix-attr:[Group(GroupLayout.GroupBox)]}
    {#ix-set:AttributeName = "<#SignalStatusWord#>"}
    CLASS AxoCtrlxDriveXscSignalStatusWord_S_0_0144_0_0
        VAR PUBLIC
            {#ix-set:AttributeName = "<#Configuration/Parametrization/Operation bit 0#>"}
            {#ix-attr:[ReadOnly()]}
            CmPmOmBit0 				:	BOOL;		//  Bit 0 of the Subdevice STM: Status, parameterization mode (S-0-0424)  !!! must be set in drive !!!
            {#ix-set:AttributeName = "<#Configuration/Parametrization/Operation bit 1#>"}
            {#ix-attr:[ReadOnly()]}
            CmPmOmBit1 				:	BOOL;		//  Bit 1 of the Subdevice STM: Status, parameterization mode (S-0-0424)  !!! must be set in drive !!!
            {#ix-set:AttributeName = "<#In target position#>"}
            {#ix-attr:[ReadOnly()]}
            InTargetPosition 				:	BOOL;		//  Bit 2 of the Positioning status: Word (S-0-0437)  !!! must be set in drive !!!
            {#ix-set:AttributeName = "<#Position command acknowledgment#>"}
            {#ix-attr:[ReadOnly()]}
            PositionCommandAck 				:	BOOL;		//  Bit 0 of the Drive-controlled positioning: Command acknowledgment (S-0-0419)  !!! must be set in drive !!!
            {#ix-set:AttributeName = "<#Drive standstill#>"}
            {#ix-attr:[ReadOnly()]}
            DriveStandstill 				:	BOOL;		//  Bit 0 of the Velocity status: Actual value = 0 (S-0-0331)  !!! must be set in drive !!!
            {#ix-set:AttributeName = "<#Command change bit#>"}
            {#ix-attr:[ReadOnly()]}
            CommandChangeBit 				:	BOOL;		//  Bit 5 of the Axis state machine: Status word, axis (P-0-0115 )  !!! must be set in drive !!!
            {#ix-set:AttributeName = "<#_bit6_Reserve#>"}
            {#ix-attr:[ReadOnly()]}
            _bit6_Reserve 				:	BOOL;
            {#ix-set:AttributeName = "<#_bit7_Reserve#>"}
            {#ix-attr:[ReadOnly()]}
            _bit7_Reserve 				:	BOOL;
            {#ix-set:AttributeName = "<#Locked by hardware#>"}
            {#ix-attr:[ReadOnly()]}
            LockedByHardware            :	BOOL;		    //  Bit 7 of the Axis state machine: Status word 2, axis (P-0-0110 )  !!! must be set in drive !!!
            {#ix-set:AttributeName = "<#_bit9_Reserve#>"}
            {#ix-attr:[ReadOnly()]}
            _bit9_Reserve 				:	BOOL;
            {#ix-set:AttributeName = "<#_bit10_Reserve#>"}
            {#ix-attr:[ReadOnly()]}
            _bit10_Reserve 				:	BOOL;
            {#ix-set:AttributeName = "<#_bit11_Reserve#>"}
            {#ix-attr:[ReadOnly()]}
            _bit11_Reserve 				:	BOOL;
            {#ix-set:AttributeName = "<#_bit12_Reserve#>"}
            {#ix-attr:[ReadOnly()]}
            _bit12_Reserve 				:	BOOL;
            {#ix-set:AttributeName = "<#_bit13_Reserve#>"}
            {#ix-attr:[ReadOnly()]}
            _bit13_Reserve 				:	BOOL;
            {#ix-set:AttributeName = "<#_bit14_Reserve#>"}
            {#ix-attr:[ReadOnly()]}
            _bit14_Reserve 				:	BOOL;
            {#ix-set:AttributeName = "<#_bit15_Reserve#>"}
            {#ix-attr:[ReadOnly()]}
            _bit15_Reserve 				:	BOOL;
        END_VAR
    END_CLASS
END_NAMESPACE

(* ---- AxoCtrlxDriveXscSupplyUnitControlWord_S_0_1720_0_1.st ---- *)
NAMESPACE AXOpen.Components.Rexroth.Drives
    {S7.extern=ReadWrite}
    {#ix-attr:[Container(Layout.Wrap)]}
    {#ix-attr:[Group(GroupLayout.GroupBox)]}
    {#ix-set:AttributeName = "<#SupplyUnitControlWord#>"}
    CLASS AxoCtrlxDriveXscSupplyUnitControlWord_S_0_1720_0_1
        VAR PUBLIC
            {#ix-set:AttributeName = "<#_bit0_Reserve#>"}
            _bit0_Reserve 				:	BOOL;
            {#ix-set:AttributeName = "<#_bit1_Reserve#>"}
            _bit1_Reserve 				:	BOOL;
            {#ix-set:AttributeName = "<#_bit2_Reserve#>"}
            _bit2_Reserve 				:	BOOL;
            {#ix-set:AttributeName = "<#_bit3_Reserve#>"}
            _bit3_Reserve 				:	BOOL;
            {#ix-set:AttributeName = "<#_bit4_Reserve#>"}
            _bit4_Reserve 				:	BOOL;
            {#ix-set:AttributeName = "<#_bit4_Reserve#>"}
            _bit5_Reserve 				:	BOOL;
            {#ix-set:AttributeName = "<#_bit6_Reserve#>"}
            _bit6_Reserve 				:	BOOL;
            {#ix-set:AttributeName = "<#_bit7_Reserve#>"}
            _bit7_Reserve 				:	BOOL;
            {#ix-set:AttributeName = "<#Mode selection bit 0#>"}
            ModeSelectionBit0 	:	BOOL;		                    //  Mode selection bit 0                                |   00:  Primary operation mode
                                                                    //                                                      |   01:  1 secondary operation mode
            {#ix-set:AttributeName = "<#Mode selection bit 1#>"}
            ModeSelectionBit1 	:	BOOL;		                    //  Command operation mode bit 1                        |   10:  2 secondary operation mode
                                                                    //                                                      |   11:  3 secondary operation mode
            {#ix-set:AttributeName = "<#DC bus discharge#>"}
            DCbusDischarge  :   BOOL;                               //  0: DC bus discharge not active
                                                                    //  1: Start DC bus discharge function
            {#ix-set:AttributeName = "<#_bit11_Reserve#>"}
            _bit11_Reserve 				:	BOOL;
            {#ix-set:AttributeName = "<#Controlling the ready for operation relay#>"}
            ControllingTheReadyForOperationRelay    :	BOOL;       //  0: Open contact
                                                                    //  1: Close contact, release
            {#ix-set:AttributeName = "<#_bit13_Reserve#>"}
            _bit13_Reserve 				:	BOOL;
            {#ix-set:AttributeName = "<#Controlling DC bus charging and mains contactor#>"}
            ControllingDCbusChargingAndMainsContactor   :	BOOL;   //  0: Mains disconnection e.g. by opening the mains contactor or by locking the mains thyristors
                                                                    //  1: Charge DC bus by closing the mains contactor or by activating the mains thyristors - device goes into rectifier mode
            {#ix-set:AttributeName = "<#Enabling#>"}
            Enabling:	BOOL;                                       //  0: Disabled, command operation mode not active
                                                                    //  1: Enabled, command operation mode active
        END_VAR
    END_CLASS
END_NAMESPACE

(* ---- AxoCtrlxDriveXscSupplyUnitStatusWord_S_0_1720_0_2.st ---- *)
NAMESPACE AXOpen.Components.Rexroth.Drives
    {S7.extern=ReadWrite}
    {#ix-attr:[Container(Layout.Wrap)]}
    {#ix-attr:[Group(GroupLayout.GroupBox)]}
    {#ix-set:AttributeName = "<#SupplyUnitStatusWord#>"}
    CLASS AxoCtrlxDriveXscSupplyUnitStatusWord_S_0_1720_0_2
        VAR PUBLIC
            {#ix-set:AttributeName = "<#_bit0_Reserve#>"}
            _bit0_Reserve 				:	BOOL;
            {#ix-set:AttributeName = "<#_bit1_Reserve#>"}
            _bit1_Reserve 				:	BOOL;
            {#ix-set:AttributeName = "<#_bit2_Reserve#>"}
            _bit2_Reserve 				:	BOOL;
            {#ix-set:AttributeName = "<#_bit3_Reserve#>"}
            _bit3_Reserve 				:	BOOL;
            {#ix-set:AttributeName = "<#Mains status#>"}
            MainsStatus				:	BOOL;
            {#ix-set:AttributeName = "<#Hardware enable#>"}
            HardwareEnable				:	BOOL;
            {#ix-set:AttributeName = "<#Controlling the mains connection#>"}
            ControllingTheMainsConnection				:	BOOL;
            {#ix-set:AttributeName = "<#Bb contact#>"}
            BbContact				:	BOOL;
            {#ix-set:AttributeName = "<#Feedback of the preselected operation modes bit 0#>"}   //  00: Primary operation mode
            PreselectedOPmodesFB_bit0    :	BOOL;                                               //  10: Secondary operation mode 2
            {#ix-set:AttributeName = "<#Feedback of the preselected operation modes bit 1#>"}   //  11: Secondary operation mode 3
            PreselectedOPmodesFB_bit01      :	BOOL;
            {#ix-set:AttributeName = "<#DC bus discharge#>"}
            DCbusDischarge  :	BOOL;
            {#ix-set:AttributeName = "<#Braking resistor#>"}
            BrakingResistor  :	BOOL;
            {#ix-set:AttributeName = "<#Warning#>"}
            Warning  :	BOOL;
            {#ix-set:AttributeName = "<#Error#>"}
            Error  :	BOOL;
            {#ix-set:AttributeName = "<#Ready for enabling#>"}
            ReadyForEnabling:	BOOL;
            {#ix-set:AttributeName = "<#Enabling#>"}
            Enabling:	BOOL;
        END_VAR
    END_CLASS
END_NAMESPACE
